FUNCTION_BLOCK StringPointerComparer EXTENDS Object IMPLEMENTS IPointerComparer
VAR
	_ClassName : STRING := __POUNAME();
END_VAR

{attribute 'monitoring' := 'call'}
PROPERTY ClassName : STRING
GET
ClassName := _ClassName;
END_GET
END_PROPERTY

{attribute "object_name" := "Compare"}
METHOD Compare : COMPARISION_RESULT
VAR_INPUT
	left : PVOID;
	right : PVOID;
END_VAR
VAR
	leftPointer : POINTER TO STRING(255); 
	rightPointer : POINTER TO STRING(255); 
END_VAR
IF left = 0 AND right = 0 THEN
	Compare := COMPARISION_RESULT.EQUALS;
	RETURN;
END_IF

IF left = 0 THEN
	Compare := COMPARISION_RESULT.LEFT_LESS_RIGHT;
	RETURN;	
END_IF

IF right = 0 THEN
	Compare := COMPARISION_RESULT.LEFT_GREATER_RIGHT;
	RETURN;	
END_IF

leftPointer := left;
rightPointer := right;

IF leftPointer^ < rightPointer^ THEN
	Compare := COMPARISION_RESULT.LEFT_LESS_RIGHT;
ELSIF leftPointer^ > rightPointer^ THEN
	Compare := COMPARISION_RESULT.LEFT_GREATER_RIGHT;
ELSE
	Compare := COMPARISION_RESULT.EQUALS;	
END_IF
END_METHOD

{attribute 'monitoring' := 'call'}
PROPERTY Size : ULINT
GET
Size := XSIZEOF(THIS^);
END_GET
END_PROPERTY

END_FUNCTION_BLOCK

(* stored: Version 1.1.0.1
   POU StringPointerComparer: Id {16d5bb33-b112-4b1b-8274-76b87c2a6e8e}, SpecialFunc None
   Property ClassName: Id {0d6be7b6-6693-44f8-9acf-8a347108c9f1}
   Get Get: Id {0c27211e-4d24-4c8f-bffc-7caca901c836}
   Method Compare: Id {430f3ac6-6207-49e3-8927-63f87475148b}
   Property Size: Id {f36ae77b-25a2-4cae-8f80-2ef698a2b05c}
   Get Get: Id {cf851a1f-6d82-4982-a1cf-a09d010101b3} *)
